Universal Robots URScript: preload4x4x3.script

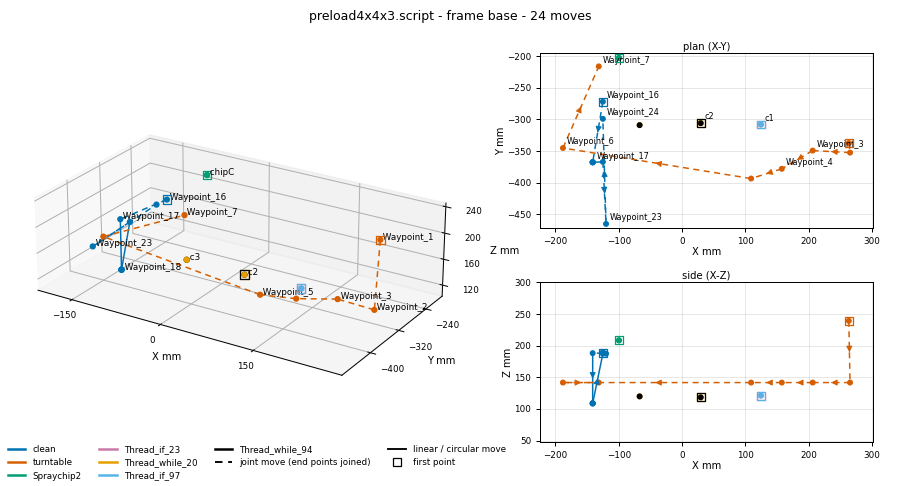
[picture p0: tool path of preload4x4x3.script in frame base, 24 of 70 moves have a stored position in this frame; points joined in program order, loops and branches not executed]
def preload4x4x3():
  global _hidden_verificationVariable=0
  step_count_fb48d3ff_0c9f_4d99_a765_ea41926c28d5 = 0.0
  thread Step_Counter_Thread_a9617a2c_6c0b_4ca4_aaba_c79477845290():
    while (True):
      step_count_fb48d3ff_0c9f_4d99_a765_ea41926c28d5 = step_count_fb48d3ff_0c9f_4d99_a765_ea41926c28d5 + 1.0
      sync()
    end
  end
  run Step_Counter_Thread_a9617a2c_6c0b_4ca4_aaba_c79477845290()
  set_standard_analog_input_domain(0, 1)
  set_standard_analog_input_domain(1, 1)
  set_tool_analog_input_domain(0, 1)
  set_tool_analog_input_domain(1, 1)
  set_analog_outputdomain(0, 0)
  set_analog_outputdomain(1, 0)
  set_input_actions_to_default()
  set_tool_communication(False, 115200, 0, 1, 1.5, 3.5)
  set_tool_output_mode(0)
  set_tool_digital_output_mode(0, 1)
  set_tool_digital_output_mode(1, 1)
  set_tool_voltage(0)
  set_safety_mode_transition_hardness(1)
  set_gravity([0.0, 0.0, 9.82])
  set_target_payload(0.530000, [0.009000, -0.039000, 0.092000], [0.000534, 0.000534, 0.000534, 0.000000, 0.000000, 0.000000])
  set_tcp(p[0.0,0.0,0.11,0.0,0.0,0.0])
  global Al_plate=p[0.12405209206180495,-0.2666666051843552,0.020008101224669964,-9.276623980477388E-5,1.8107917580596192E-5,3.1233857134705927]
  global Frame2x2=p[0.18266245434305164,-0.34273121659514855,0.026002571110600767,-2.225423529876215E-4,3.0110667546023537E-4,3.1233976058306383]
  global Plane_1=p[0.0,0.0,0.0,0.0,0.0,0.0]
  global URlogoTutorial=p[-0.08178353973148575,-0.3363174165299142,0.04788621506469384,-3.9746155723688456E-5,-3.4682148779121894E-5,-1.5668291789091222]
  global carousel=p[0.13865255139760183,-0.25132593351268107,0.051531504137083003,-4.453572132438073E-5,-1.3071222590669835E-4,-3.1349676625391965]
  global carouselrod=p[0.2020731702281844,-0.34951442511341274,0.1947611446273096,3.139766958234101,-0.10689428010274801,-1.1796370330365635E-5]
  global paper=p[-0.09670794781244417,-0.3283412964648025,0.027665994240809913,-3.2057893450593004E-5,2.867088716161181E-5,-1.6085327915291054]
  global rod=p[0.13368013097420872,-0.41123185103490206,0.09926814901395645,2.2214229924093103,-2.2214158162465862,-2.9165882738638143E-5]
  global timer_1=0
  global c1_p=p[.124631079723, -.308028756414, .121202819455, -3.141124231191, .028500472376, .002927495869]
  global c1_q=[-0.7796428839312952, -1.6496883831419886, -1.8346924781799316, -1.2288200122169037, 1.571037769317627, 3.949756145477295]
  global c2_p=p[.029526817192, -.305921948164, .118391903226, -3.141181649485, .028353160101, .002761019314]
  global c2_q=[-1.032529656087057, -1.5420829218677063, -1.959731101989746, -1.2109692853740235, 1.5706452131271362, 3.6968348026275635]
  global c3_p=p[-.067038459763, -.309045591369, .119904708816, -3.141192610771, .028366655788, .002743930455]
  global c3_q=[-1.3553932348834437, -1.5796953640379847, -1.9152411222457886, -1.2173438531211396, 1.570389747619629, 3.3739569187164307]
  global Waypoint_16_p=p[-.125097928533, -.271984222044, .188211676824, -3.139810722578, .105446315311, .000070958927]
  global Waypoint_16_q=[-1.5480602423297327, -1.4491210740855713, -1.7099264860153198, -1.552596167927124, 1.5715936422348022, 3.23006010055542]
  global Waypoint_17_p=p[-.141183217597, -.367684006591, .188213447751, 3.139821760490, -.105397104768, -.000067867997]
  global Waypoint_17_q=[-1.597567383443014, -1.8740092716612757, -1.241610050201416, -1.5960084400572718, 1.5719740390777588, 3.1803600788116455]
  global Waypoint_18_p=p[-.141178244459, -.367687282910, .108904454765, 3.139816402425, -.105408093734, -.000060814483]
  global Waypoint_18_q=[-1.5975983778582972, -1.9245020351805628, -1.550661325454712, -1.2364590925029297, 1.5723340511322021, 3.1807193756103516]
  global Waypoint_19_p=p[-.141189357305, -.367687267469, .108915260822, 3.121780755938, .351957921543, -.000099281586]
  global Waypoint_19_q=[-1.5976179281817835, -1.9244748554625453, -1.550661325454712, -1.2364507478526612, 1.572314977645874, 2.889045000076294]
  global Waypoint_20_p=p[-.141176698746, -.367682773595, .108907204798, -3.111042719163, .436975672702, .000063164110]
  global Waypoint_20_q=[-1.5975945631610315, -1.9244939289488734, -1.5506495237350464, -1.2365017098239441, 1.5723340511322021, 3.3926987648010254]
  global Waypoint_21_p=p[-.141174078526, -.367696805030, .108909057026, 3.139786221315, -.105395786134, -.000060564502]
  global Waypoint_21_q=[-1.597586456929342, -1.9245058498778285, -1.5506460666656494, -1.2364399594119568, 1.5723340511322021, 3.1807241439819336]
  global Waypoint_22_p=p[-.125093999497, -.367099400456, .187371407622, 3.139783011421, -.105392168035, -.000053869150]
  global Waypoint_22_q=[-1.5538747946368616, -1.846323629418844, -1.2822730541229248, -1.5829936466612757, 1.5719654560089111, 3.224064588546753]
  global Waypoint_23_p=p[-.120064390322, -.465070651334, .187365924664, 2.700279766902, -.088400420341, .019763045538]
  global Waypoint_23_q=[-1.5412524382220667, -1.9475652180113734, -1.406833291053772, -0.9173591893962403, 1.5603561401367188, 3.2332537174224854]
  global Waypoint_24_p=p[-.125099110421, -.299097154487, .189878767902, 3.139750209928, -.105401717856, -.000111797080]
  global Waypoint_24_q=[-1.550074879323141, -1.5617311683348198, -1.5979981422424316, -1.5518303674510499, 1.5716702938079834, 3.2279696464538574]
  global Waypoint_1_p=p[.263501689877, -.337317763427, .239349489480, 3.139797243720, -.105347053477, -.000037720516]
  global Waypoint_1_q=[-0.5959728399859827, -2.1057659588255824, -0.6533136367797852, -1.9525557957091273, 1.5718059539794922, 4.181682586669922]
  global Waypoint_2_p=p[.265438435610, -.352444474661, .141740907029, 3.139726376264, -.105360108121, -.000022031768]
  global Waypoint_2_q=[-0.6231134573565882, -2.1016999683775843, -1.126999020576477, -1.4828875821879883, 1.5722739696502686, 4.154912948608398]
  global Waypoint_3_p=p[.206441973084, -.349241721273, .141737893294, 3.139734184252, -.105329347268, -.000022485776]
  global Waypoint_3_q=[-0.7073677221881312, -1.9410401783385218, -1.3681066036224365, -1.4024366003325959, 1.5721865892410278, 4.070710182189941]
  global Waypoint_4_p=p[.157616611756, -.378012026932, .141738203587, 3.139764187573, -.105376653239, -.000076760662]
  global Waypoint_4_q=[-0.8494070211993616, -1.9579774341978968, -1.3439116477966309, -1.409730003481247, 1.5722019672393799, 3.928692579269409]
  global Waypoint_5_p=p[.109134761588, -.393436595889, .141742225598, 3.139732501163, -.105376381431, -.000050533951]
  global Waypoint_5_q=[-0.972816292439596, -1.9523960552611292, -1.3519116640090942, -1.4072665137103577, 1.5721949338912964, 3.805286407470703]
  global Waypoint_6_p=p[-.188131250090, -.345166366147, .141750553976, 3.139727051239, -.105353578209, -.000024875816]
  global Waypoint_6_q=[-1.7293437162982386, -1.8864180050291957, -1.4439769983291626, -1.381135032778122, 1.572224736213684, 3.0487747192382812]
  global Waypoint_7_p=p[-.131564048097, -.216205376465, .141741700579, 3.139714533984, -.105382776464, -.000044168049]
  global Waypoint_7_q=[-1.572542969380514, -1.2417927545360108, -2.0833356380462646, -1.3863917154124756, 1.571577787399292, 3.2058310508728027]
  global chipC_p=p[-.099703384862, -.202952364142, .208439850600, 3.139657619359, -.105437397760, -.000145108772]
  global chipC_q=[-1.4082325140582483, -1.0998719197562714, -1.8470008373260498, -1.7646123371519984, 1.5710017681121826, 3.3699307441711426]
  global Waypoint_15_p=p[-.099704296715, -.202951379992, .208432580258, 3.139670120847, -.105426183766, -.000160358536]
  global Waypoint_15_q=[-1.4082286993609827, -1.099871740942337, -1.8470300436019897, -1.764597078362936, 1.5709946155548096, 3.369927167892456]
  global timer_1_is_counting=False
  thread Timer_Thread():
    while (True):
      if (timer_1_is_counting):
        timer_1 = timer_1 + get_steptime()
      end
      sync()
    end
  end
  run Timer_Thread()
  def CircleAllangles():
    $ 266 "CircleAllangles" "noBreak"
    $ 267 "p0≔p[c[0]+r,c[1],c[2],c[3],c[4],c[5]-1.5*A]"
    global p0=p[c[0]+r,c[1],c[2],c[3],c[4],c[5]-1.5*A]
    $ 268 "p45≔p[c[0]+0.71*r,c[1]+0.71*r,c[2],c[3]-A/1.1,c[4],c[5]-A/1.1]"
    global p45=p[c[0]+0.71*r,c[1]+0.71*r,c[2],c[3]-A/1.1,c[4],c[5]-A/1.1]
    $ 269 "p90≔p[c[0],c[1]+r,c[2],c[3]-A,c[4],c[5]]"
    global p90=p[c[0],c[1]+r,c[2],c[3]-A,c[4],c[5]]
    $ 270 "p135≔p[c[0]-0.71*r,c[1]+0.71*r,c[2],c[3]-A/1.1,c[4],c[5]+A/1.1]"
    global p135=p[c[0]-0.71*r,c[1]+0.71*r,c[2],c[3]-A/1.1,c[4],c[5]+A/1.1]
    $ 271 "p180≔p[c[0]-r,c[1],c[2],c[3],c[4],c[5]+1.5*A]"
    global p180=p[c[0]-r,c[1],c[2],c[3],c[4],c[5]+1.5*A]
    $ 272 "p225≔p[c[0]-0.71*r,c[1]-0.71*r,c[2],c[3]+A/1.1,c[4],c[5]+A/1.1]"
    global p225=p[c[0]-0.71*r,c[1]-0.71*r,c[2],c[3]+A/1.1,c[4],c[5]+A/1.1]
    $ 273 "p270≔p[c[0],c[1]-r,c[2],c[3]+A,c[4],c[5]]"
    global p270=p[c[0],c[1]-r,c[2],c[3]+A,c[4],c[5]]
    $ 274 "p315≔p[c[0]+0.71*r,c[1]-0.71*r,c[2],c[3]+A/1.1,c[4],c[5]-A/1.1]"
    global p315=p[c[0]+0.71*r,c[1]-0.71*r,c[2],c[3]+A/1.1,c[4],c[5]-A/1.1]
    $ 275 "Set atomization=On"
    set_standard_digital_out(1, True)
    $ 276 "Set triggersolenoid=On"
    set_standard_digital_out(0, True)
    $ 277 "MoveL"
    $ 278 "p0" "breakAfter"
    set_tcp(p[0.0,0.0,0.11,0.0,0.0,0.0])
    movel(p0, a=1.3, v=0.4, r=0.005)
    $ 279 "p45" "breakAfter"
    set_tcp(p[0.0,0.0,0.11,0.0,0.0,0.0])
    movel(p45, a=1.3, v=0.4, r=0.005)
    $ 280 "p90" "breakAfter"
    set_tcp(p[0.0,0.0,0.11,0.0,0.0,0.0])
    movel(p90, a=1.3, v=0.4, r=0.005)
    $ 281 "p135" "breakAfter"
    set_tcp(p[0.0,0.0,0.11,0.0,0.0,0.0])
    movel(p135, a=1.3, v=0.4, r=0.005)
    $ 282 "p180" "breakAfter"
    set_tcp(p[0.0,0.0,0.11,0.0,0.0,0.0])
    movel(p180, a=1.3, v=0.4, r=0.005)
    $ 283 "p225" "breakAfter"
    set_tcp(p[0.0,0.0,0.11,0.0,0.0,0.0])
    movel(p225, a=1.3, v=0.4, r=0.005)
    $ 284 "p270" "breakAfter"
    set_tcp(p[0.0,0.0,0.11,0.0,0.0,0.0])
    movel(p270, a=1.3, v=0.4, r=0.005)
    $ 285 "p315" "breakAfter"
    set_tcp(p[0.0,0.0,0.11,0.0,0.0,0.0])
    movel(p315, a=1.3, v=0.4, r=0.005)
    $ 286 "p0" "breakAfter"
    set_tcp(p[0.0,0.0,0.11,0.0,0.0,0.0])
    movel(p0, a=1.3, v=0.4, r=0.005)
    $ 287 "p45" "breakAfter"
    set_tcp(p[0.0,0.0,0.11,0.0,0.0,0.0])
    movel(p45, a=1.3, v=0.4, r=0.005)
    $ 288 "p90" "breakAfter"
    set_tcp(p[0.0,0.0,0.11,0.0,0.0,0.0])
    movel(p90, a=1.3, v=0.4, r=0.005)
    $ 289 "Set atomization=Off"
    set_standard_digital_out(1, False)
    $ 290 "Set triggersolenoid=Off"
    set_standard_digital_out(0, False)
  end
  def clean():
    $ 291 "clean" "noBreak"
    $ 292 "MoveJ"
    $ 293 "Waypoint_16" "breakAfter"
    movej(get_inverse_kin(Waypoint_16_p, qnear=Waypoint_16_q), a=1.3962634015954636, v=1.0471975511965976)
    $ 294 "Waypoint_17" "breakAfter"
    movej(get_inverse_kin(Waypoint_17_p, qnear=Waypoint_17_q), a=1.3962634015954636, v=1.0471975511965976)
    $ 295 "MoveL"
    $ 296 "Waypoint_18" "breakAfter"
    movel(Waypoint_18_p, a=1.2, v=0.05)
    $ 297 "MoveL"
    $ 298 "Waypoint_19" "breakAfter"
    movel(Waypoint_19_p, a=1.2, v=0.05)
    $ 299 "MoveL"
    $ 300 "Waypoint_20" "breakAfter"
    movel(Waypoint_20_p, a=1.2, v=0.05)
    $ 301 "MoveL"
    $ 302 "Waypoint_21" "breakAfter"
    movel(Waypoint_21_p, a=1.2, v=0.05)
    $ 303 "MoveL"
    $ 304 "Waypoint_22" "breakAfter"
    movel(Waypoint_22_p, a=1.2, v=0.25)
    $ 305 "MoveJ"
    $ 306 "Waypoint_23" "breakAfter"
    movej(get_inverse_kin(Waypoint_23_p, qnear=Waypoint_23_q), a=1.3962634015954636, v=1.0471975511965976)
    $ 307 "Set atomization=On"
    set_standard_digital_out(1, True)
    $ 308 "Set triggersolenoid=On"
    set_standard_digital_out(0, True)
    $ 309 "Wait: 0.2"
    sleep(0.2)
    $ 310 "Set atomization=Off"
    set_standard_digital_out(1, False)
    $ 311 "Set triggersolenoid=Off"
    set_standard_digital_out(0, False)
    $ 312 "MoveJ"
    $ 313 "Waypoint_24" "breakAfter"
    movej(get_inverse_kin(Waypoint_24_p, qnear=Waypoint_24_q), a=1.3962634015954636, v=1.0471975511965976)
  end
  def turntable():
    $ 314 "turntable" "noBreak"
    $ 315 "MoveJ"
    $ 316 "Waypoint_1" "breakAfter"
    set_tcp(p[0.0,0.0,0.11,0.0,0.0,0.0])
    movej(get_inverse_kin(pose_trans(carouselrod, pose_trans(p[-.225374943892, -.334963115579, .194760490892, -3.139766958285, .106894280104, .000011796367], Waypoint_1_p)), qnear=Waypoint_1_q), a=1.3962634015954636, v=0.5235987755982988, r=0.02)
    $ 317 "Waypoint_2" "breakAfter"
    set_tcp(p[0.0,0.0,0.11,0.0,0.0,0.0])
    movej(get_inverse_kin(pose_trans(carouselrod, pose_trans(p[-.225374943892, -.334963115579, .194760490892, -3.139766958285, .106894280104, .000011796367], Waypoint_2_p)), qnear=Waypoint_2_q), a=1.3962634015954636, v=0.5235987755982988, r=0.02)
    $ 318 "Waypoint_3" "breakAfter"
    set_tcp(p[0.0,0.0,0.11,0.0,0.0,0.0])
    movej(get_inverse_kin(pose_trans(carouselrod, pose_trans(p[-.225374943892, -.334963115579, .194760490892, -3.139766958285, .106894280104, .000011796367], Waypoint_3_p)), qnear=Waypoint_3_q), a=1.3962634015954636, v=0.5235987755982988, r=0.02)
    $ 319 "Waypoint_4" "breakAfter"
    set_tcp(p[0.0,0.0,0.11,0.0,0.0,0.0])
    movej(get_inverse_kin(pose_trans(carouselrod, pose_trans(p[-.225374943892, -.334963115579, .194760490892, -3.139766958285, .106894280104, .000011796367], Waypoint_4_p)), qnear=Waypoint_4_q), a=1.3962634015954636, v=0.5235987755982988, r=0.02)
    $ 320 "Waypoint_5" "breakAfter"
    set_tcp(p[0.0,0.0,0.11,0.0,0.0,0.0])
    movej(get_inverse_kin(pose_trans(carouselrod, pose_trans(p[-.225374943892, -.334963115579, .194760490892, -3.139766958285, .106894280104, .000011796367], Waypoint_5_p)), qnear=Waypoint_5_q), a=1.3962634015954636, v=0.5235987755982988, r=0.02)
    $ 321 "MoveJ"
    $ 322 "Waypoint_6" "breakAfter"
    movej(get_inverse_kin(pose_trans(carouselrod, pose_trans(p[-.225374943892, -.334963115579, .194760490892, -3.139766958285, .106894280104, .000011796367], Waypoint_6_p)), qnear=Waypoint_6_q), a=1.3962634015954636, v=0.3141592653589793)
    $ 323 "Wait: 1.0"
    sleep(1.0)
    $ 324 "MoveJ"
    $ 325 "Waypoint_7" "breakAfter"
    movej(get_inverse_kin(pose_trans(carouselrod, pose_trans(p[-.225374943892, -.334963115579, .194760490892, -3.139766958285, .106894280104, .000011796367], Waypoint_7_p)), qnear=Waypoint_7_q), a=1.3962634015954636, v=1.0471975511965976, r=0.02)
  end
  def Spraychip2():
    $ 326 "Spraychip2" "noBreak"
    $ 327 "MoveJ"
    $ 328 "chipC" "breakAfter"
    movej(get_inverse_kin(chipC_p, qnear=chipC_q), a=1.3962634015954636, v=1.0471975511965976)
    $ 329 "c≔chipC"
    global c=chipC_p
    $ 330 "rc≔27/1000"
    global rc=27/1000
    $ 331 "p0≔p[c[0]+rc,c[1],c[2],c[3],c[4],c[5]-1.5*0]"
    global p0=p[c[0]+rc,c[1],c[2],c[3],c[4],c[5]-1.5*0]
    $ 332 "p45≔p[c[0]+0.71*rc,c[1]+0.71*rc,c[2],c[3]-0/1.1,c[4],c[5]-0/1.1]"
    global p45=p[c[0]+0.71*rc,c[1]+0.71*rc,c[2],c[3]-0/1.1,c[4],c[5]-0/1.1]
    $ 333 "p90≔p[c[0],c[1]+rc,c[2],c[3]-0,c[4],c[5]]"
    global p90=p[c[0],c[1]+rc,c[2],c[3]-0,c[4],c[5]]
    $ 334 "p135≔p[c[0]-0.71*rc,c[1]+0.71*rc,c[2],c[3]-0/1.1,c[4],c[5]+0/1.1]"
    global p135=p[c[0]-0.71*rc,c[1]+0.71*rc,c[2],c[3]-0/1.1,c[4],c[5]+0/1.1]
    $ 335 "p180≔p[c[0]-rc,c[1],c[2],c[3],c[4],c[5]+1.5*0]"
    global p180=p[c[0]-rc,c[1],c[2],c[3],c[4],c[5]+1.5*0]
    $ 336 "p225≔p[c[0]-0.71*rc,c[1]-0.71*rc,c[2],c[3]+0/1.1,c[4],c[5]+0/1.1]"
    global p225=p[c[0]-0.71*rc,c[1]-0.71*rc,c[2],c[3]+0/1.1,c[4],c[5]+0/1.1]
    $ 337 "p270≔p[c[0],c[1]-rc,c[2],c[3]+0,c[4],c[5]]"
    global p270=p[c[0],c[1]-rc,c[2],c[3]+0,c[4],c[5]]
    $ 338 "p315≔p[c[0]+0.71*rc,c[1]-0.71*rc,c[2],c[3]+0/1.1,c[4],c[5]-0/1.1]"
    global p315=p[c[0]+0.71*rc,c[1]-0.71*rc,c[2],c[3]+0/1.1,c[4],c[5]-0/1.1]
    $ 339 "Set atomization=On"
    set_standard_digital_out(1, True)
    $ 340 "Set triggersolenoid=On"
    set_standard_digital_out(0, True)
    $ 341 "MoveL"
    $ 342 "p0" "breakAfter"
    set_tcp(p[0.0,0.0,0.11,0.0,0.0,0.0])
    movel(p0, a=1.3, v=0.085, r=0.01)
    $ 343 "p45" "breakAfter"
    set_tcp(p[0.0,0.0,0.11,0.0,0.0,0.0])
    movel(p45, a=1.3, v=0.085, r=0.01)
    $ 344 "p90" "breakAfter"
    set_tcp(p[0.0,0.0,0.11,0.0,0.0,0.0])
    movel(p90, a=1.3, v=0.085, r=0.01)
    $ 345 "p135" "breakAfter"
    set_tcp(p[0.0,0.0,0.11,0.0,0.0,0.0])
    movel(p135, a=1.3, v=0.085, r=0.01)
    $ 346 "p180" "breakAfter"
    set_tcp(p[0.0,0.0,0.11,0.0,0.0,0.0])
    movel(p180, a=1.3, v=0.085, r=0.01)
    $ 347 "Set triggersolenoid=Off"
    set_standard_digital_out(0, False)
    $ 348 "Wait: 0.1"
    sleep(0.1)
    $ 349 "Set triggersolenoid=On"
    set_standard_digital_out(0, True)
    $ 350 "p225" "breakAfter"
    set_tcp(p[0.0,0.0,0.11,0.0,0.0,0.0])
    movel(p225, a=1.3, v=0.085, r=0.01)
    $ 351 "p270" "breakAfter"
    set_tcp(p[0.0,0.0,0.11,0.0,0.0,0.0])
    movel(p270, a=1.3, v=0.085, r=0.01)
    $ 352 "p315" "breakAfter"
    set_tcp(p[0.0,0.0,0.11,0.0,0.0,0.0])
    movel(p315, a=1.3, v=0.085, r=0.01)
    $ 353 "p0" "breakAfter"
    set_tcp(p[0.0,0.0,0.11,0.0,0.0,0.0])
    movel(p0, a=1.3, v=0.085, r=0.01)
    $ 354 "p45" "breakAfter"
    set_tcp(p[0.0,0.0,0.11,0.0,0.0,0.0])
    movel(p45, a=1.3, v=0.085, r=0.01)
    $ 355 "Set triggersolenoid=Off"
    set_standard_digital_out(0, False)
    $ 356 "Wait: 0.1"
    sleep(0.1)
    $ 357 "Set triggersolenoid=On"
    set_standard_digital_out(0, True)
    $ 358 "p90" "breakAfter"
    set_tcp(p[0.0,0.0,0.11,0.0,0.0,0.0])
    movel(p90, a=1.3, v=0.085, r=0.01)
    $ 359 "p135" "breakAfter"
    set_tcp(p[0.0,0.0,0.11,0.0,0.0,0.0])
    movel(p135, a=1.3, v=0.085, r=0.01)
    $ 360 "p180" "breakAfter"
    set_tcp(p[0.0,0.0,0.11,0.0,0.0,0.0])
    movel(p180, a=1.3, v=0.085, r=0.01)
    $ 361 "p225" "breakAfter"
    set_tcp(p[0.0,0.0,0.11,0.0,0.0,0.0])
    movel(p225, a=1.3, v=0.085, r=0.01)
    $ 362 "p270" "breakAfter"
    set_tcp(p[0.0,0.0,0.11,0.0,0.0,0.0])
    movel(p270, a=1.3, v=0.085, r=0.01)
    $ 363 "p315" "breakAfter"
    set_tcp(p[0.0,0.0,0.11,0.0,0.0,0.0])
    movel(p315, a=1.3, v=0.085, r=0.01)
    $ 364 "p0" "breakAfter"
    set_tcp(p[0.0,0.0,0.11,0.0,0.0,0.0])
    movel(p0, a=1.3, v=0.085, r=0.01)
    $ 365 "MoveJ"
    $ 366 "Waypoint_15" "breakAfter"
    movej(get_inverse_kin(Waypoint_15_p, qnear=Waypoint_15_q), a=1.3962634015954636, v=1.0471975511965976)
    $ 367 "Wait: 0.2"
    sleep(0.2)
    $ 368 "Set atomization=Off"
    set_standard_digital_out(1, False)
    $ 369 "Set triggersolenoid=Off"
    set_standard_digital_out(0, False)
  end
  while (True):
    $ 2 "Robot Program"
    $ 3 "'Program to be used for part #124517-055 SRF preload'"
    # 'Program to be used for part #124517-055 SRF preload'
    $ 4 "'Program rev ___: mm/dd/yy note'"
    # 'Program rev ___: mm/dd/yy note'
    $ 5 "timer_1: Start"
    timer_1_is_counting = True
    $ 6 "r≔1/1000"
    global r=1/1000
    $ 7 "A≔8*3.1416/180"
    global A=8*3.1416/180
    $ 10 "sidenum≔3"
    global sidenum=3
    $ 12 "coatnum≔2"
    global coatnum=2
    $ 14 "partnum≔2"
    global partnum=2
    $ 15 "Loop_1≔1"
    global Loop_1=1
    $ 16 "If partnum≤sidenum"
    global thread_flag_16=0
    thread Thread_if_16():
      $ 17 "Loop (coatnum)>0"
      thread Thread_while_17():
        while (True):
          $ 18 "partleft≔partnum"
          global partleft=partnum
          $ 19 "loopnum≔1"
          global loopnum=1
          $ 20 "Loop partleft>0"
          thread Thread_while_20():
            while (True):
              $ 21 "Call clean"
              clean()
              $ 22 "Call Spraychip2"
              Spraychip2()
              $ 23 "If loopnum≟1 or loopnum≟4 or loopnum≟7 or loopnum≟10"
              global thread_flag_23=0
              thread Thread_if_23():
                $ 24 "MoveJ"
                $ 25 "c1" "breakAfter"
                movej(get_inverse_kin(c1_p, qnear=c1_q), a=1.3962634015954636, v=1.0471975511965976)
                $ 26 "c≔c1"
                global c=c1_p
                $ 27 "Call CircleAllangles"
                CircleAllangles()
                $ 28 "x2≔p[c[0]-0.037,c[1],c[2],c[3],c[4],c[5]]"
                global x2=p[c[0]-0.037,c[1],c[2],c[3],c[4],c[5]]
                $ 29 "x3≔p[c[0]-0.037,c[1]+0.037,c[2],c[3],c[4],c[5]]"
                global x3=p[c[0]-0.037,c[1]+0.037,c[2],c[3],c[4],c[5]]
                $ 30 "x4≔p[c[0],c[1]+0.037,c[2],c[3],c[4],c[5]]"
                global x4=p[c[0],c[1]+0.037,c[2],c[3],c[4],c[5]]
                $ 31 "MoveJ"
                $ 32 "x2" "breakAfter"
                movej(x2, a=1.3962634015954636, v=1.0471975511965976)
                $ 33 "c≔x2"
                global c=x2
                $ 34 "Call CircleAllangles"
                CircleAllangles()
                $ 35 "MoveJ"
                $ 36 "x3" "breakAfter"
                movej(x3, a=1.3962634015954636, v=1.0471975511965976)
                $ 37 "c≔x3"
                global c=x3
                $ 38 "Call CircleAllangles"
                CircleAllangles()
                $ 39 "MoveJ"
                $ 40 "x4" "breakAfter"
                movej(x4, a=1.3962634015954636, v=1.0471975511965976)
                $ 41 "c≔x4"
                global c=x4
                $ 42 "Call CircleAllangles"
                CircleAllangles()
                thread_flag_23 = 1
              end
              if (loopnum == 1  or  loopnum == 4  or  loopnum == 7  or  loopnum == 10):
                global thread_handler_23=run Thread_if_23()
                while (thread_flag_23 == 0):
                  if not(loopnum == 1  or  loopnum == 4  or  loopnum == 7  or  loopnum == 10):
                    kill thread_handler_23
                    thread_flag_23 = 2
                  else:
                    sync()
                  end
                end
              else:
                thread_flag_23 = 2
              end
              if (thread_flag_23 == 2):
                $ 43 "ElseIf loopnum≟2 or loopnum≟5 or loopnum≟8 or loopnum≟11"
                if (loopnum == 2  or  loopnum == 5  or  loopnum == 8  or  loopnum == 11):
                  $ 44 "MoveJ"
                  $ 45 "c2" "breakAfter"
                  movej(get_inverse_kin(c2_p, qnear=c2_q), a=1.3962634015954636, v=1.0471975511965976)
                  $ 46 "c≔c2"
                  global c=c2_p
                  $ 47 "Call CircleAllangles"
                  CircleAllangles()
                  $ 48 "x2≔p[c[0]-0.037,c[1],c[2],c[3],c[4],c[5]]"
                  global x2=p[c[0]-0.037,c[1],c[2],c[3],c[4],c[5]]
                  $ 49 "x3≔p[c[0]-0.037,c[1]+0.037,c[2],c[3],c[4],c[5]]"
                  global x3=p[c[0]-0.037,c[1]+0.037,c[2],c[3],c[4],c[5]]
                  $ 50 "x4≔p[c[0],c[1]+0.037,c[2],c[3],c[4],c[5]]"
                  global x4=p[c[0],c[1]+0.037,c[2],c[3],c[4],c[5]]
                  $ 51 "MoveJ"
                  $ 52 "x2" "breakAfter"
                  movej(x2, a=1.3962634015954636, v=1.0471975511965976)
                  $ 53 "c≔x2"
                  global c=x2
                  $ 54 "Call CircleAllangles"
                  CircleAllangles()
                  $ 55 "MoveJ"
                  $ 56 "x3" "breakAfter"
                  movej(x3, a=1.3962634015954636, v=1.0471975511965976)
                  $ 57 "c≔x3"
                  global c=x3
                  $ 58 "Call CircleAllangles"
                  CircleAllangles()
                  $ 59 "MoveJ"
                  $ 60 "x4" "breakAfter"
                  movej(x4, a=1.3962634015954636, v=1.0471975511965976)
                  $ 61 "c≔x4"
                  global c=x4
                  $ 62 "Call CircleAllangles"
                  CircleAllangles()
                else:
                  $ 63 "Else" "noBreak"
                  $ 64 "MoveJ"
                  $ 65 "c3" "breakAfter"
                  movej(get_inverse_kin(c3_p, qnear=c3_q), a=1.3962634015954636, v=1.0471975511965976)
                  $ 66 "c≔c3"
                  global c=c3_p
                  $ 67 "Call CircleAllangles"
                  CircleAllangles()
                  $ 68 "x2≔p[c[0]-0.037,c[1],c[2],c[3],c[4],c[5]]"
                  global x2=p[c[0]-0.037,c[1],c[2],c[3],c[4],c[5]]
                  $ 69 "x3≔p[c[0]-0.037,c[1]+0.037,c[2],c[3],c[4],c[5]]"
                  global x3=p[c[0]-0.037,c[1]+0.037,c[2],c[3],c[4],c[5]]
                  $ 70 "x4≔p[c[0],c[1]+0.037,c[2],c[3],c[4],c[5]]"
                  global x4=p[c[0],c[1]+0.037,c[2],c[3],c[4],c[5]]
                  $ 71 "MoveJ"
                  $ 72 "x2" "breakAfter"
                  movej(x2, a=1.3962634015954636, v=1.0471975511965976)
                  $ 73 "c≔x2"
                  global c=x2
                  $ 74 "Call CircleAllangles"
                  CircleAllangles()
                  $ 75 "MoveJ"
                  $ 76 "x3" "breakAfter"
                  movej(x3, a=1.3962634015954636, v=1.0471975511965976)
                  $ 77 "c≔x3"
                  global c=x3
                  $ 78 "Call CircleAllangles"
                  CircleAllangles()
                  $ 79 "MoveJ"
                  $ 80 "x4" "breakAfter"
                  movej(x4, a=1.3962634015954636, v=1.0471975511965976)
                  $ 81 "c≔x4"
                  global c=x4
                  $ 82 "Call CircleAllangles"
                  CircleAllangles()
                  $ 83 "Wait: 4.0"
                  sleep(4.0)
                end
              end
              $ 84 "loopnum≔loopnum+1"
              global loopnum=loopnum+1
              $ 85 "partleft≔partleft-1"
              global partleft=partleft-1
            end
          end
          if (partleft>0):
            global thread_handler_20=run Thread_while_20()
            while (partleft>0):
              sync()
            end
            kill thread_handler_20
          end
          $ 86 "i≔0"
          global i=0
          $ 87 "coatnum≔coatnum-1"
          global coatnum=coatnum-1
        end
      end
      if ((coatnum)>0):
        global thread_handler_17=run Thread_while_17()
        while ((coatnum)>0):
          sync()
        end
        kill thread_handler_17
      end
      $ 88 "Halt"
      halt
      thread_flag_16 = 1
    end
    if (partnum <= sidenum):
      global thread_handler_16=run Thread_if_16()
      while (thread_flag_16 == 0):
        if not(partnum <= sidenum):
          kill thread_handler_16
          thread_flag_16 = 2
        else:
          sync()
        end
      end
    else:
      thread_flag_16 = 2
    end
    if (thread_flag_16 == 2):
      $ 89 "Else" "noBreak"
      $ 90 "Loop (coatnum)>0"
      thread Thread_while_90():
        while (True):
          $ 91 "partleft≔partnum"
          global partleft=partnum
          $ 92 "loopnum≔1"
          global loopnum=1
          $ 93 "turnnum≔0"
          global turnnum=0
          $ 94 "Loop partleft>0"
          thread Thread_while_94():
            while (True):
              $ 95 "Call clean"
              clean()
              $ 96 "Call Spraychip2"
              Spraychip2()
              $ 97 "If loopnum≟1 or loopnum≟4 or loopnum≟7 or loopnum≟10"
              global thread_flag_97=0
              thread Thread_if_97():
                $ 98 "MoveJ"
                $ 99 "c1" "breakAfter"
                movej(get_inverse_kin(c1_p, qnear=c1_q), a=1.3962634015954636, v=1.0471975511965976)
                $ 100 "c≔c1"
                global c=c1_p
                $ 101 "Call CircleAllangles"
                CircleAllangles()
                $ 102 "x2≔p[c[0]-0.037,c[1],c[2],c[3],c[4],c[5]]"
                global x2=p[c[0]-0.037,c[1],c[2],c[3],c[4],c[5]]
                $ 103 "x3≔p[c[0]-0.037,c[1]+0.037,c[2],c[3],c[4],c[5]]"
                global x3=p[c[0]-0.037,c[1]+0.037,c[2],c[3],c[4],c[5]]
                $ 104 "x4≔p[c[0],c[1]+0.037,c[2],c[3],c[4],c[5]]"
                global x4=p[c[0],c[1]+0.037,c[2],c[3],c[4],c[5]]
                $ 105 "MoveJ"
                $ 106 "x2" "breakAfter"
                movej(x2, a=1.3962634015954636, v=1.0471975511965976)
                $ 107 "c≔x2"
                global c=x2
                $ 108 "Call CircleAllangles"
                CircleAllangles()
                $ 109 "MoveJ"
                $ 110 "x3" "breakAfter"
                movej(x3, a=1.3962634015954636, v=1.0471975511965976)
                $ 111 "c≔x3"
                global c=x3
                $ 112 "Call CircleAllangles"
                CircleAllangles()
                $ 113 "MoveJ"
                $ 114 "x4" "breakAfter"
                movej(x4, a=1.3962634015954636, v=1.0471975511965976)
                $ 115 "c≔x4"
                global c=x4
                $ 116 "Call CircleAllangles"
                CircleAllangles()
                thread_flag_97 = 1
              end
              if (loopnum == 1  or  loopnum == 4  or  loopnum == 7  or  loopnum == 10):
                global thread_handler_97=run Thread_if_97()
                while (thread_flag_97 == 0):
                  if not(loopnum == 1  or  loopnum == 4  or  loopnum == 7  or  loopnum == 10):
                    kill thread_handler_97
                    thread_flag_97 = 2
                  else:
                    sync()
                  end
                end
              else:
                thread_flag_97 = 2
              end
              if (thread_flag_97 == 2):
                $ 117 "ElseIf loopnum≟2 or loopnum≟5 or loopnum≟8 or loopnum≟11"
                if (loopnum == 2  or  loopnum == 5  or  loopnum == 8  or  loopnum == 11):
                  $ 118 "MoveJ"
                  $ 119 "c2" "breakAfter"
                  movej(get_inverse_kin(c2_p, qnear=c2_q), a=1.3962634015954636, v=1.0471975511965976)
                  $ 120 "c≔c2"
                  global c=c2_p
                  $ 121 "Call CircleAllangles"
                  CircleAllangles()
                  $ 122 "x2≔p[c[0]-0.037,c[1],c[2],c[3],c[4],c[5]]"
                  global x2=p[c[0]-0.037,c[1],c[2],c[3],c[4],c[5]]
                  $ 123 "x3≔p[c[0]-0.037,c[1]+0.037,c[2],c[3],c[4],c[5]]"
                  global x3=p[c[0]-0.037,c[1]+0.037,c[2],c[3],c[4],c[5]]
                  $ 124 "x4≔p[c[0],c[1]+0.037,c[2],c[3],c[4],c[5]]"
                  global x4=p[c[0],c[1]+0.037,c[2],c[3],c[4],c[5]]
                  $ 125 "MoveJ"
                  $ 126 "x2" "breakAfter"
                  movej(x2, a=1.3962634015954636, v=1.0471975511965976)
                  $ 127 "c≔x2"
                  global c=x2
                  $ 128 "Call CircleAllangles"
                  CircleAllangles()
                  $ 129 "MoveJ"
                  $ 130 "x3" "breakAfter"
                  movej(x3, a=1.3962634015954636, v=1.0471975511965976)
                  $ 131 "c≔x3"
                  global c=x3
                  $ 132 "Call CircleAllangles"
                  CircleAllangles()
                  $ 133 "MoveJ"
                  $ 134 "x4" "breakAfter"
                  movej(x4, a=1.3962634015954636, v=1.0471975511965976)
                  $ 135 "c≔x4"
                  global c=x4
                  $ 136 "Call CircleAllangles"
                  CircleAllangles()
                else:
                  $ 137 "Else" "noBreak"
                  $ 138 "MoveJ"
                  $ 139 "c3" "breakAfter"
                  movej(get_inverse_kin(c3_p, qnear=c3_q), a=1.3962634015954636, v=1.0471975511965976)
                  $ 140 "c≔c3"
                  global c=c3_p
                  $ 141 "Call CircleAllangles"
                  CircleAllangles()
                  $ 142 "x2≔p[c[0]-0.037,c[1],c[2],c[3],c[4],c[5]]"
                  global x2=p[c[0]-0.037,c[1],c[2],c[3],c[4],c[5]]
                  $ 143 "x3≔p[c[0]-0.037,c[1]+0.037,c[2],c[3],c[4],c[5]]"
                  global x3=p[c[0]-0.037,c[1]+0.037,c[2],c[3],c[4],c[5]]
                  $ 144 "x4≔p[c[0],c[1]+0.037,c[2],c[3],c[4],c[5]]"
                  global x4=p[c[0],c[1]+0.037,c[2],c[3],c[4],c[5]]
                  $ 145 "MoveJ"
                  $ 146 "x2" "breakAfter"
                  movej(x2, a=1.3962634015954636, v=1.0471975511965976)
                  $ 147 "c≔x2"
                  global c=x2
                  $ 148 "Call CircleAllangles"
                  CircleAllangles()
                  $ 149 "MoveJ"
                  $ 150 "x3" "breakAfter"
                  movej(x3, a=1.3962634015954636, v=1.0471975511965976)
                  $ 151 "c≔x3"
                  global c=x3
                  $ 152 "Call CircleAllangles"
                  CircleAllangles()
                  $ 153 "MoveJ"
                  $ 154 "x4" "breakAfter"
                  movej(x4, a=1.3962634015954636, v=1.0471975511965976)
                  $ 155 "c≔x4"
                  global c=x4
                  $ 156 "Call CircleAllangles"
                  CircleAllangles()
                  $ 157 "Wait: 4.0"
                  sleep(4.0)
                end
              end
              $ 158 "loopnum≔loopnum+1"
              global loopnum=loopnum+1
              $ 159 "partleft≔partleft-1"
              global partleft=partleft-1
            end
          end
          if (partleft>0):
            global thread_handler_94=run Thread_while_94()
            while (partleft>0):
              sync()
            end
            kill thread_handler_94
          end
          $ 160 "i≔0"
          global i=0
          $ 161 "Loop (6-turnnum)>0"
          thread Thread_while_161():
            while (True):
              $ 162 "Call turntable"
              turntable()
              $ 163 "turnnum≔turnnum+1"
              global turnnum=turnnum+1
            end
          end
          if ((6-turnnum)>0):
            global thread_handler_161=run Thread_while_161()
            while ((6-turnnum)>0):
              sync()
            end
            kill thread_handler_161
          end
          $ 164 "coatnum≔coatnum-1"
          global coatnum=coatnum-1
        end
      end
      if ((coatnum)>0):
        global thread_handler_90=run Thread_while_90()
        while ((coatnum)>0):
          sync()
        end
        kill thread_handler_90
      end
      $ 165 "Halt"
      halt
    end
  end
end
